# EPICS IOC start-up script: iocsh/ethercatmcAxisdebug.iocsh
dbLoadRecords("ethercatmcdebug.template", "PREFIX=$(PREFIX), AXIS_NAME=$(AXIS_NAME), MOTOR_PORT=$(MOTOR_PORT), AXIS_NO=$(AXIS_NO), PREC=3")
